PROGRAM MAIN
VAR
	iState 		: INT 	:= 0;	
	iMethod		: SINT 	:= 0;
	
	bCreateContainer	: 	BOOL := FALSE;
	bRemoveContainer	:	BOOL := FALSE;
	
	
	bSensorLagerUnten		: BOOL;
	bSensorLagerMitte		: BOOL; 
	
	
	fbSeperator		: FB_Separator;
	staSep			: State;
	instVereinzelung : Model_Seperator;
	
	temp	: BOOL := FALSE;
	enzSens1 : BOOL;
	enzSens2 : BOOL;
	enzSens3 : BOOL;
END_VAR

// Call models	
instVereinzelung(
	ssMethodType:= iMethod, Signal_CreateContainer:= bCreateContainer, 	c_Signal_RemoveContainerOnC:= bRemoveContainer, 
	SamplingTime:= 0.005, 
	Hw_AktObenEinfahren:= IFC_HW.R1AKT1,	// einfahren
 	Hw_AktObenAusfahren:= IFC_HW.R2AKT1,	// ausfahren
	Hw_AktUntenEinfahren:= IFC_HW.R2AKT2,	// einfahren
 	Hw_AktUntenAusfahren:= IFC_HW.R1AKT2, 	// ausfahren
	Signal_Storage2=> bSensorLagerMitte,
 	Signal_Storage1=> bSensorLagerUnten, 
	Hw_SensorOben=> enzSens3,
 	Hw_SensorMitte=> enzSens2,
 	Hw_SensorUnten=> enzSens1);
IFC_HW.EinzelSens1 := enzSens1;
IFC_HW.EinzelSens2 := enzSens2;
IFC_HW.EinzelSens3 := enzSens3;

	
// Call Functionblocks
fbSeperator(
	bEnable:= TRUE, bExecute:= temp, bErrorReset:= , 
	bSensor1:= IFC_HW.EinzelSens1,
 	bSensor2:= IFC_HW.EinzelSens2,
 	bSensor3:= IFC_HW.EinzelSens3, 
	bR1AKT1=> IFC_HW.R1AKT1,	// einfahren
 	bR2AKT1=> IFC_HW.R2AKT1,	// ausfahren
 	bR1AKT2=> IFC_HW.R1AKT2,	// ausfahren
 	bR2AKT2=> IFC_HW.R2AKT2, 	// einfahren
	bNoBottle=> IFC_HW.NoBottle, 
	bWrongBottle=> IFC_HW.WrongBottle, 
	eStatus=> staSep);	

	
// Visualization Inventor
IFC_HW.Inv_Vereinz_Container1 := BOOL_TO_REAL(IFC_HW.EinzelSens1);
IFC_HW.Inv_Vereinz_Container2 := BOOL_TO_REAL(IFC_HW.EinzelSens2);
IFC_HW.Inv_Vereinz_Container3 := BOOL_TO_REAL(IFC_HW.EinzelSens3);
IFC_HW.Inv_Vereinz_Container4 := BOOL_TO_REAL(bSensorLagerUnten);
IFC_HW.Inv_Vereinz_Container5 := BOOL_TO_REAL(bSensorLagerMitte);

IF (IFC_HW.R1AKT1 = TRUE) THEN 
	IFC_HW.Inv_Vereinz_HubmagnetOben := 1;
ELSIF (IFC_HW.R2AKT1 = TRUE) THEN
	IFC_HW.Inv_Vereinz_HubmagnetOben := 0;
END_IF

IF (IFC_HW.R2AKT2 = TRUE) THEN
	IFC_HW.Inv_Vereinz_HubmagnetUnten := 1;
ELSIF (IFC_HW.R1AKT2 = TRUE) THEN
	IFC_HW.Inv_Vereinz_HubmagnetUnten := 0;
END_IF



//AdsVariables.HubmagnetOben_ADS := BOOL_TO_REAL(bHubmagnetOben);
//AdsVariables.HubmagnetUnten_ADS := BOOL_TO_REAL(bHubmagnetUnten);
	



// State Machine
CASE iState OF
	0:
		
		iState := iState +1;
	1:
		iMethod := 1;
END_CASE

END_PROGRAM

(* stored: Version 1.1.0.1, ProductVersion 3.1.4024.10
   POU MAIN: Id {fef2700b-e0b1-4384-91dc-030dd6cbb394}, SpecialFunc None *)
